// TIA Portal V15.1 export
// export: Created 2024-05-17T05:38:54.5333761Z, ExportSetting WithDefaults, DisplayName Totally Integrated Automation Portal, DisplayVersion V15.1 Update 5, DisplayName TIA Portal Openness, DisplayVersion V15.1 Update 5, DisplayName SINAMICS Startdrive Advanced, DisplayVersion V15.1, DisplayName G130, G150, S120, S150, SINAMICS MV, S210, DisplayVersion V15.1, DisplayName G110M, G120, G120C, G120D, G120P, DisplayVersion V15.1, DisplayName STEP 7 Professional, DisplayVersion V15.1 Update 5, DisplayName STEP 7 Safety, DisplayVersion V15.1, DisplayName WinCC Professional, DisplayVersion V15.1 Update 5, DisplayName SIMATIC Visualization Architect, DisplayVersion V15.1
FUNCTION "209220ZS01Passiv" : Void   // FC373, FBD
TITLE = 209220ZS01Passiv
{ S7_Optimized_Access := 'FALSE' }
AUTHOR : VCC
NAME : LocFunc
VERSION : 0.1
// stored: AutoNumber false, IsIECCheckEnabled false, SetENOAutomatically False, UDAEnableTagReadback false
   VAR_OUTPUT
      O_AlarmA : Bool;   // Alarm A
      O_AlarmB : Bool;   // Alarm B
      O_AlarmC : Bool;   // Alarm C
      O_AlarmD : Bool;   // Alarm D
      O_AlarmABCondition : Bool;   // Alarms resetable
      H_IAnim : Word;   // Icon Animation
   END_VAR
   VAR_TEMP
      TEMP0 : Bool;
   END_VAR
BEGIN

REGION Network 1: **** --------------------- ET200sp I/O --------------------- ****
END_REGION

REGION Network 2: **** 2.2 - Alarms - Alarm Generation **** 209000AK04JX37QF5270 - ET200sp I/O - Safety Card QF5270
   // Passivation alarm - ET200sp I/O - Safety Card QF5270
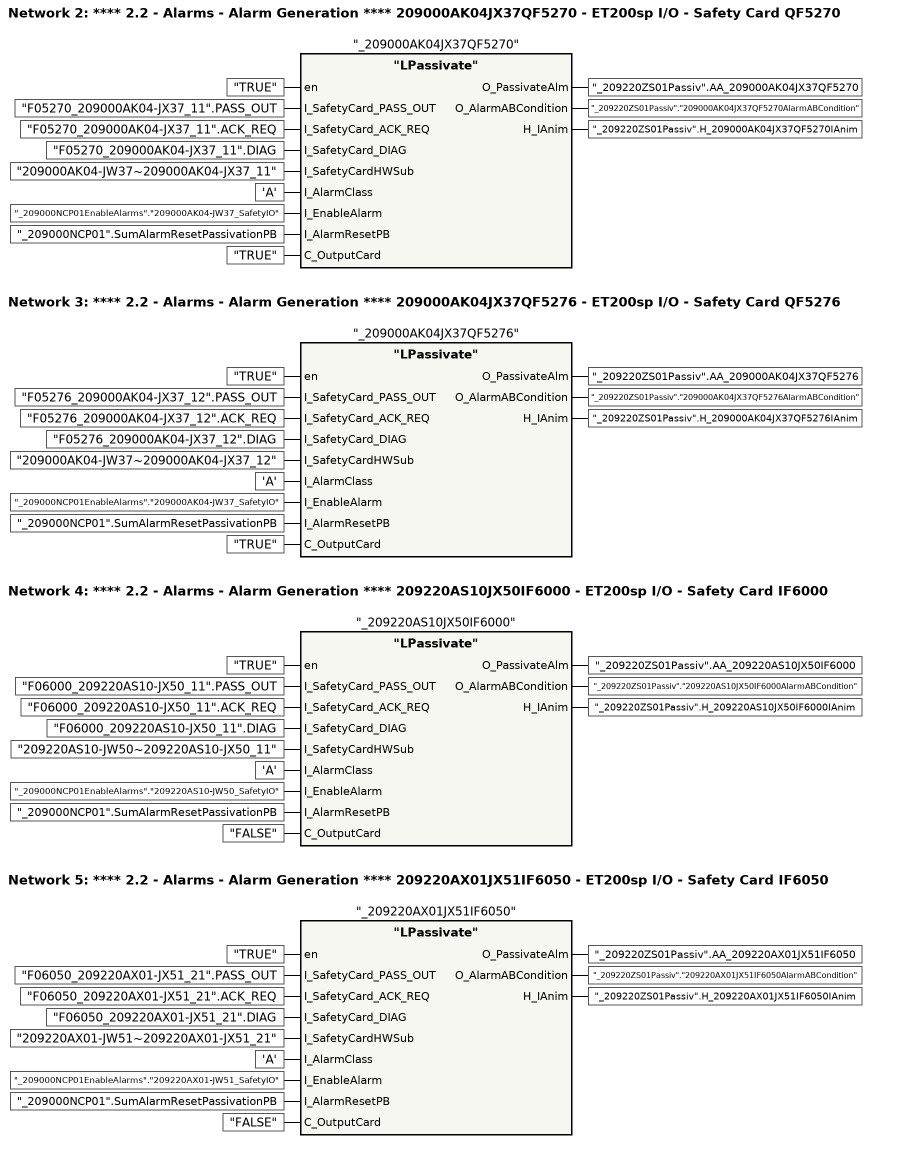
   IF "TRUE" THEN
       "_209000AK04JX37QF5270"(I_SafetyCard_PASS_OUT := "F05270_209000AK04-JX37_11".PASS_OUT,   // "LPassivate"
                               I_SafetyCard_ACK_REQ := "F05270_209000AK04-JX37_11".ACK_REQ,
                               I_SafetyCard_DIAG := "F05270_209000AK04-JX37_11".DIAG,
                               I_SafetyCardHWSub := "209000AK04-JW37~209000AK04-JX37_11",
                               I_AlarmClass := 'A',
                               I_EnableAlarm := "_209000NCP01EnableAlarms"."209000AK04-JW37_SafetyIO",
                               I_AlarmResetPB := "_209000NCP01".SumAlarmResetPassivationPB,
                               C_OutputCard := "TRUE",
                               O_PassivateAlm => "_209220ZS01Passiv".AA_209000AK04JX37QF5270,
                               O_AlarmABCondition => "_209220ZS01Passiv"."209000AK04JX37QF5270AlarmABCondition",
                               H_IAnim => "_209220ZS01Passiv".H_209000AK04JX37QF5270IAnim);
   END_IF;
END_REGION

REGION Network 3: **** 2.2 - Alarms - Alarm Generation **** 209000AK04JX37QF5276 - ET200sp I/O - Safety Card QF5276
   // Passivation alarm - ET200sp I/O - Safety Card QF5276
   IF "TRUE" THEN
       "_209000AK04JX37QF5276"(I_SafetyCard_PASS_OUT := "F05276_209000AK04-JX37_12".PASS_OUT,   // "LPassivate"
                               I_SafetyCard_ACK_REQ := "F05276_209000AK04-JX37_12".ACK_REQ,
                               I_SafetyCard_DIAG := "F05276_209000AK04-JX37_12".DIAG,
                               I_SafetyCardHWSub := "209000AK04-JW37~209000AK04-JX37_12",
                               I_AlarmClass := 'A',
                               I_EnableAlarm := "_209000NCP01EnableAlarms"."209000AK04-JW37_SafetyIO",
                               I_AlarmResetPB := "_209000NCP01".SumAlarmResetPassivationPB,
                               C_OutputCard := "TRUE",
                               O_PassivateAlm => "_209220ZS01Passiv".AA_209000AK04JX37QF5276,
                               O_AlarmABCondition => "_209220ZS01Passiv"."209000AK04JX37QF5276AlarmABCondition",
                               H_IAnim => "_209220ZS01Passiv".H_209000AK04JX37QF5276IAnim);
   END_IF;
END_REGION

REGION Network 4: **** 2.2 - Alarms - Alarm Generation **** 209220AS10JX50IF6000 - ET200sp I/O - Safety Card IF6000
   // Passivation alarm - ET200sp I/O - Safety Card IF6000
   IF "TRUE" THEN
       "_209220AS10JX50IF6000"(I_SafetyCard_PASS_OUT := "F06000_209220AS10-JX50_11".PASS_OUT,   // "LPassivate"
                               I_SafetyCard_ACK_REQ := "F06000_209220AS10-JX50_11".ACK_REQ,
                               I_SafetyCard_DIAG := "F06000_209220AS10-JX50_11".DIAG,
                               I_SafetyCardHWSub := "209220AS10-JW50~209220AS10-JX50_11",
                               I_AlarmClass := 'A',
                               I_EnableAlarm := "_209000NCP01EnableAlarms"."209220AS10-JW50_SafetyIO",
                               I_AlarmResetPB := "_209000NCP01".SumAlarmResetPassivationPB,
                               C_OutputCard := "FALSE",
                               O_PassivateAlm => "_209220ZS01Passiv".AA_209220AS10JX50IF6000,
                               O_AlarmABCondition => "_209220ZS01Passiv"."209220AS10JX50IF6000AlarmABCondition",
                               H_IAnim => "_209220ZS01Passiv".H_209220AS10JX50IF6000IAnim);
   END_IF;
END_REGION

REGION Network 5: **** 2.2 - Alarms - Alarm Generation **** 209220AX01JX51IF6050 - ET200sp I/O - Safety Card IF6050
   // Passivation alarm - ET200sp I/O - Safety Card IF6050
   IF "TRUE" THEN
       "_209220AX01JX51IF6050"(I_SafetyCard_PASS_OUT := "F06050_209220AX01-JX51_21".PASS_OUT,   // "LPassivate"
                               I_SafetyCard_ACK_REQ := "F06050_209220AX01-JX51_21".ACK_REQ,
                               I_SafetyCard_DIAG := "F06050_209220AX01-JX51_21".DIAG,
                               I_SafetyCardHWSub := "209220AX01-JW51~209220AX01-JX51_21",
                               I_AlarmClass := 'A',
                               I_EnableAlarm := "_209000NCP01EnableAlarms"."209220AX01-JW51_SafetyIO",
                               I_AlarmResetPB := "_209000NCP01".SumAlarmResetPassivationPB,
                               C_OutputCard := "FALSE",
                               O_PassivateAlm => "_209220ZS01Passiv".AA_209220AX01JX51IF6050,
                               O_AlarmABCondition => "_209220ZS01Passiv"."209220AX01JX51IF6050AlarmABCondition",
                               H_IAnim => "_209220ZS01Passiv".H_209220AX01JX51IF6050IAnim);
   END_IF;
END_REGION

REGION Network 6: **** 2.2 - Alarms - Alarm Generation **** 209220AS11JX52IF6100 - ET200sp I/O - Safety Card IF6100
   // Passivation alarm - ET200sp I/O - Safety Card IF6100
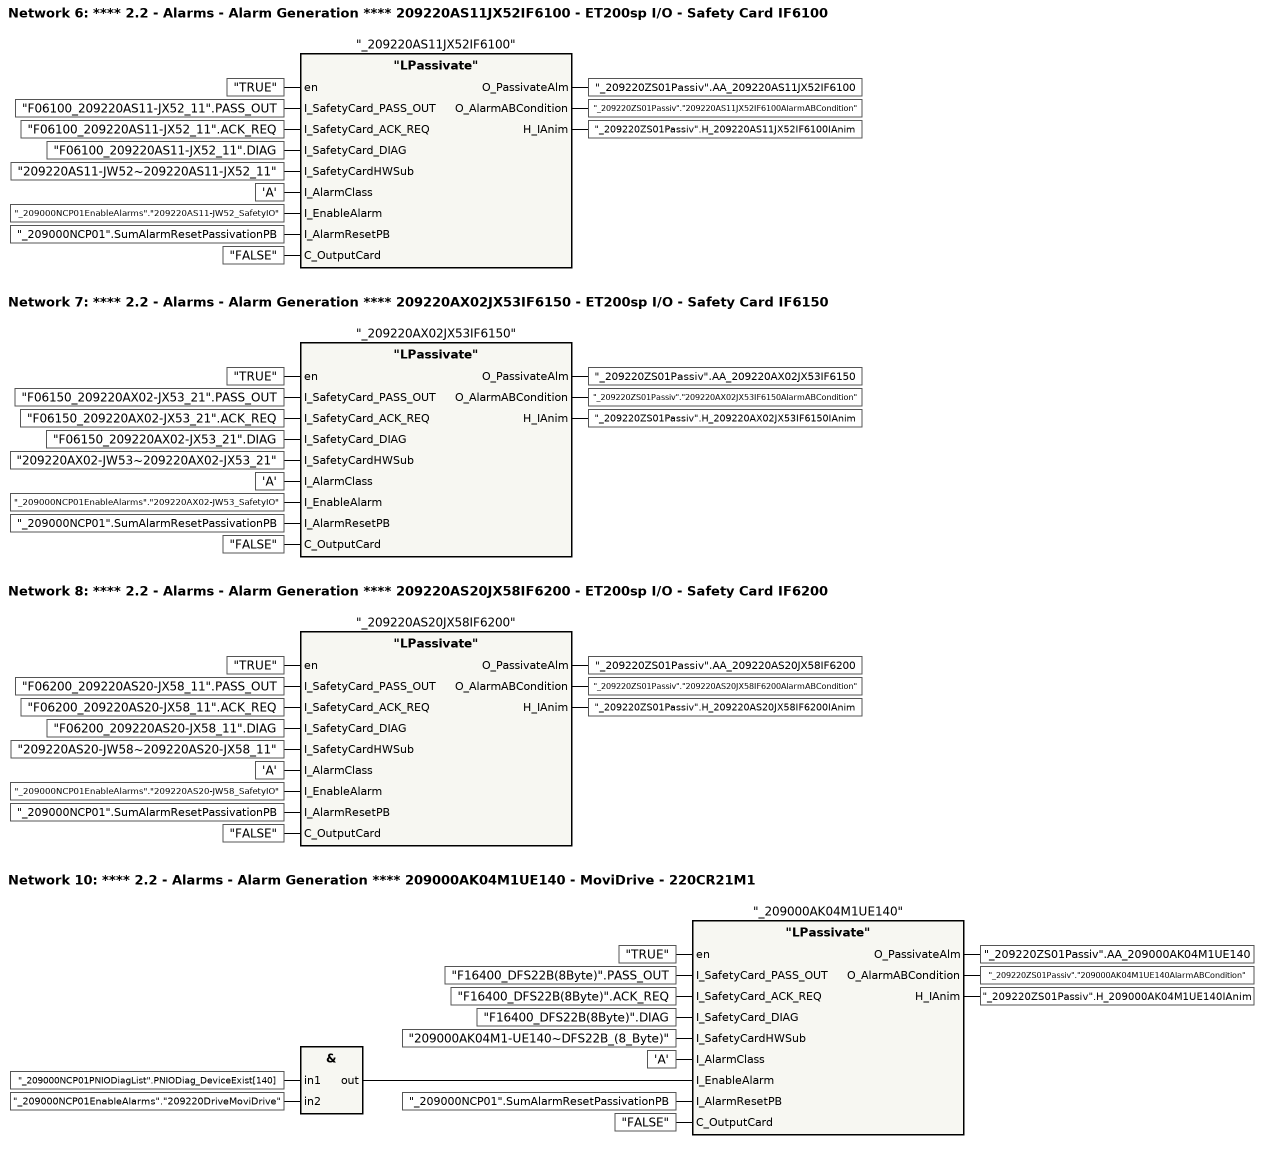
   IF "TRUE" THEN
       "_209220AS11JX52IF6100"(I_SafetyCard_PASS_OUT := "F06100_209220AS11-JX52_11".PASS_OUT,   // "LPassivate"
                               I_SafetyCard_ACK_REQ := "F06100_209220AS11-JX52_11".ACK_REQ,
                               I_SafetyCard_DIAG := "F06100_209220AS11-JX52_11".DIAG,
                               I_SafetyCardHWSub := "209220AS11-JW52~209220AS11-JX52_11",
                               I_AlarmClass := 'A',
                               I_EnableAlarm := "_209000NCP01EnableAlarms"."209220AS11-JW52_SafetyIO",
                               I_AlarmResetPB := "_209000NCP01".SumAlarmResetPassivationPB,
                               C_OutputCard := "FALSE",
                               O_PassivateAlm => "_209220ZS01Passiv".AA_209220AS11JX52IF6100,
                               O_AlarmABCondition => "_209220ZS01Passiv"."209220AS11JX52IF6100AlarmABCondition",
                               H_IAnim => "_209220ZS01Passiv".H_209220AS11JX52IF6100IAnim);
   END_IF;
END_REGION

REGION Network 7: **** 2.2 - Alarms - Alarm Generation **** 209220AX02JX53IF6150 - ET200sp I/O - Safety Card IF6150
   // Passivation alarm - ET200sp I/O - Safety Card IF6150
   IF "TRUE" THEN
       "_209220AX02JX53IF6150"(I_SafetyCard_PASS_OUT := "F06150_209220AX02-JX53_21".PASS_OUT,   // "LPassivate"
                               I_SafetyCard_ACK_REQ := "F06150_209220AX02-JX53_21".ACK_REQ,
                               I_SafetyCard_DIAG := "F06150_209220AX02-JX53_21".DIAG,
                               I_SafetyCardHWSub := "209220AX02-JW53~209220AX02-JX53_21",
                               I_AlarmClass := 'A',
                               I_EnableAlarm := "_209000NCP01EnableAlarms"."209220AX02-JW53_SafetyIO",
                               I_AlarmResetPB := "_209000NCP01".SumAlarmResetPassivationPB,
                               C_OutputCard := "FALSE",
                               O_PassivateAlm => "_209220ZS01Passiv".AA_209220AX02JX53IF6150,
                               O_AlarmABCondition => "_209220ZS01Passiv"."209220AX02JX53IF6150AlarmABCondition",
                               H_IAnim => "_209220ZS01Passiv".H_209220AX02JX53IF6150IAnim);
   END_IF;
END_REGION

REGION Network 8: **** 2.2 - Alarms - Alarm Generation **** 209220AS20JX58IF6200 - ET200sp I/O - Safety Card IF6200
   // Passivation alarm - ET200sp I/O - Safety Card IF6200
   IF "TRUE" THEN
       "_209220AS20JX58IF6200"(I_SafetyCard_PASS_OUT := "F06200_209220AS20-JX58_11".PASS_OUT,   // "LPassivate"
                               I_SafetyCard_ACK_REQ := "F06200_209220AS20-JX58_11".ACK_REQ,
                               I_SafetyCard_DIAG := "F06200_209220AS20-JX58_11".DIAG,
                               I_SafetyCardHWSub := "209220AS20-JW58~209220AS20-JX58_11",
                               I_AlarmClass := 'A',
                               I_EnableAlarm := "_209000NCP01EnableAlarms"."209220AS20-JW58_SafetyIO",
                               I_AlarmResetPB := "_209000NCP01".SumAlarmResetPassivationPB,
                               C_OutputCard := "FALSE",
                               O_PassivateAlm => "_209220ZS01Passiv".AA_209220AS20JX58IF6200,
                               O_AlarmABCondition => "_209220ZS01Passiv"."209220AS20JX58IF6200AlarmABCondition",
                               H_IAnim => "_209220ZS01Passiv".H_209220AS20JX58IF6200IAnim);
   END_IF;
END_REGION

REGION Network 9: **** --------------------- Drive --------------------- ****
END_REGION

REGION Network 10: **** 2.2 - Alarms - Alarm Generation **** 209000AK04M1UE140 - MoviDrive - 220CR21M1
   // Passivation alarm - MoviDrive - 220CR21M1
   IF "TRUE" THEN
       "_209000AK04M1UE140"(I_SafetyCard_PASS_OUT := "F16400_DFS22B(8Byte)".PASS_OUT,   // "LPassivate"
                            I_SafetyCard_ACK_REQ := "F16400_DFS22B(8Byte)".ACK_REQ,
                            I_SafetyCard_DIAG := "F16400_DFS22B(8Byte)".DIAG,
                            I_SafetyCardHWSub := "209000AK04M1-UE140~DFS22B_(8_Byte)",
                            I_AlarmClass := 'A',
                            I_EnableAlarm := "_209000NCP01PNIODiagList".PNIODiag_DeviceExist[140] AND "_209000NCP01EnableAlarms"."209220DriveMoviDrive",
                            I_AlarmResetPB := "_209000NCP01".SumAlarmResetPassivationPB,
                            C_OutputCard := "FALSE",
                            O_PassivateAlm => "_209220ZS01Passiv".AA_209000AK04M1UE140,
                            O_AlarmABCondition => "_209220ZS01Passiv"."209000AK04M1UE140AlarmABCondition",
                            H_IAnim => "_209220ZS01Passiv".H_209000AK04M1UE140IAnim);
   END_IF;
END_REGION

REGION Network 11: **** 2.2 - Alarms - Alarm Generation **** 209000AK04M4UE141 - MoviDrive - 220CS22M4ME1 (Power)
   // Passivation alarm - MoviDrive - 220CS22M4ME1 (Power)
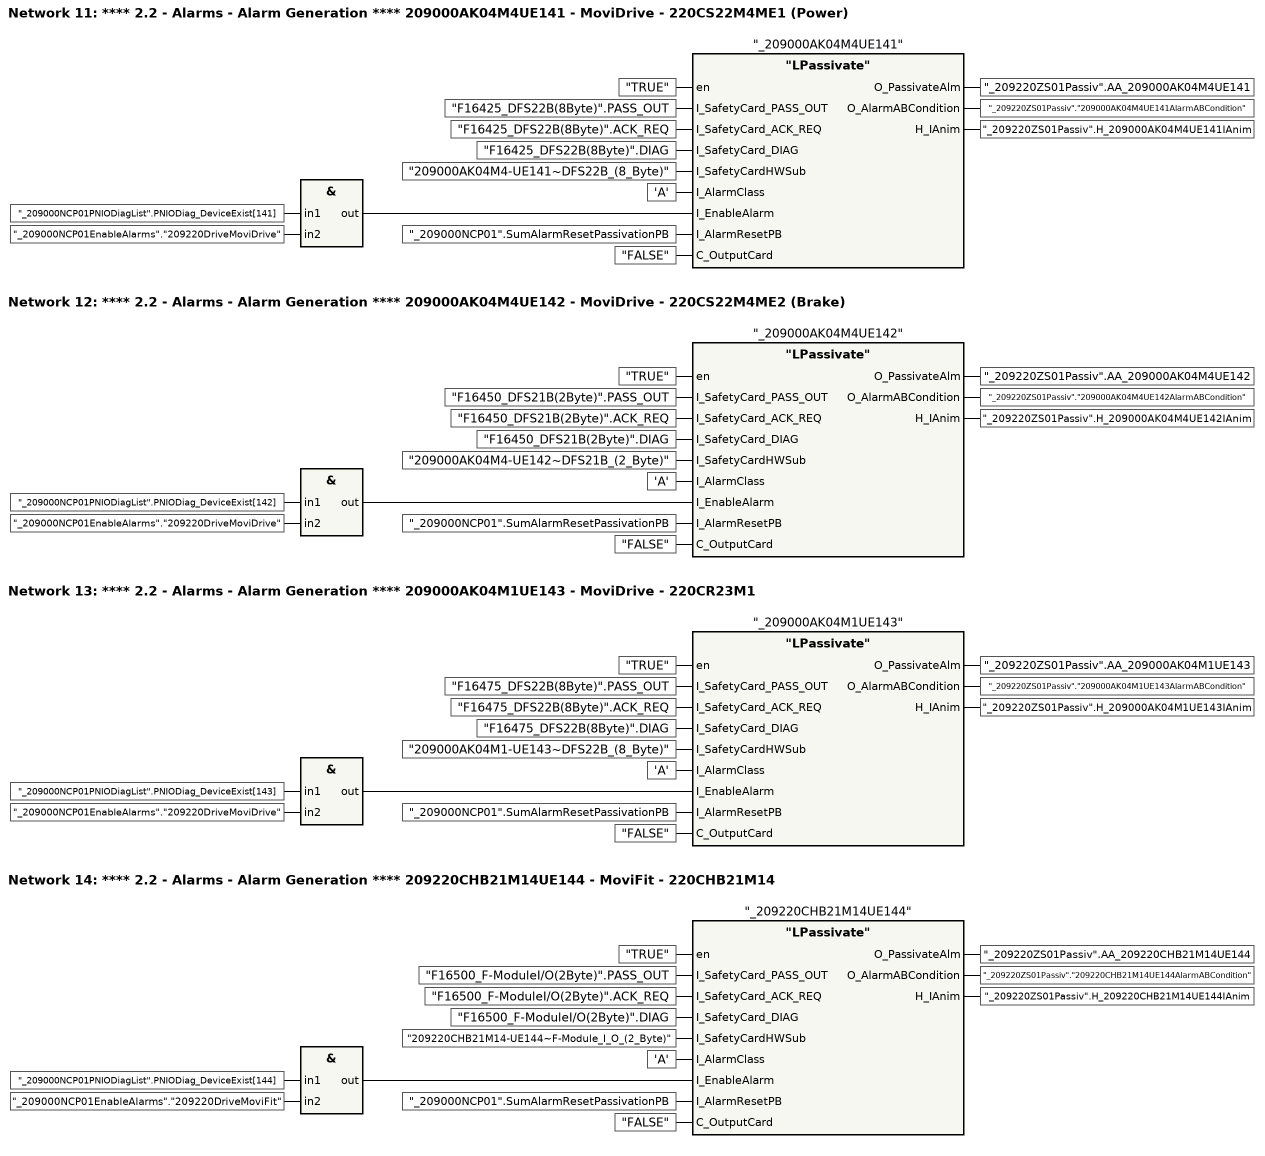
   IF "TRUE" THEN
       "_209000AK04M4UE141"(I_SafetyCard_PASS_OUT := "F16425_DFS22B(8Byte)".PASS_OUT,   // "LPassivate"
                            I_SafetyCard_ACK_REQ := "F16425_DFS22B(8Byte)".ACK_REQ,
                            I_SafetyCard_DIAG := "F16425_DFS22B(8Byte)".DIAG,
                            I_SafetyCardHWSub := "209000AK04M4-UE141~DFS22B_(8_Byte)",
                            I_AlarmClass := 'A',
                            I_EnableAlarm := "_209000NCP01PNIODiagList".PNIODiag_DeviceExist[141] AND "_209000NCP01EnableAlarms"."209220DriveMoviDrive",
                            I_AlarmResetPB := "_209000NCP01".SumAlarmResetPassivationPB,
                            C_OutputCard := "FALSE",
                            O_PassivateAlm => "_209220ZS01Passiv".AA_209000AK04M4UE141,
                            O_AlarmABCondition => "_209220ZS01Passiv"."209000AK04M4UE141AlarmABCondition",
                            H_IAnim => "_209220ZS01Passiv".H_209000AK04M4UE141IAnim);
   END_IF;
END_REGION

REGION Network 12: **** 2.2 - Alarms - Alarm Generation **** 209000AK04M4UE142 - MoviDrive - 220CS22M4ME2 (Brake)
   // Passivation alarm - MoviDrive - 220CS22M4ME2 (Brake)
   IF "TRUE" THEN
       "_209000AK04M4UE142"(I_SafetyCard_PASS_OUT := "F16450_DFS21B(2Byte)".PASS_OUT,   // "LPassivate"
                            I_SafetyCard_ACK_REQ := "F16450_DFS21B(2Byte)".ACK_REQ,
                            I_SafetyCard_DIAG := "F16450_DFS21B(2Byte)".DIAG,
                            I_SafetyCardHWSub := "209000AK04M4-UE142~DFS21B_(2_Byte)",
                            I_AlarmClass := 'A',
                            I_EnableAlarm := "_209000NCP01PNIODiagList".PNIODiag_DeviceExist[142] AND "_209000NCP01EnableAlarms"."209220DriveMoviDrive",
                            I_AlarmResetPB := "_209000NCP01".SumAlarmResetPassivationPB,
                            C_OutputCard := "FALSE",
                            O_PassivateAlm => "_209220ZS01Passiv".AA_209000AK04M4UE142,
                            O_AlarmABCondition => "_209220ZS01Passiv"."209000AK04M4UE142AlarmABCondition",
                            H_IAnim => "_209220ZS01Passiv".H_209000AK04M4UE142IAnim);
   END_IF;
END_REGION

REGION Network 13: **** 2.2 - Alarms - Alarm Generation **** 209000AK04M1UE143 - MoviDrive - 220CR23M1
   // Passivation alarm - MoviDrive - 220CR23M1
   IF "TRUE" THEN
       "_209000AK04M1UE143"(I_SafetyCard_PASS_OUT := "F16475_DFS22B(8Byte)".PASS_OUT,   // "LPassivate"
                            I_SafetyCard_ACK_REQ := "F16475_DFS22B(8Byte)".ACK_REQ,
                            I_SafetyCard_DIAG := "F16475_DFS22B(8Byte)".DIAG,
                            I_SafetyCardHWSub := "209000AK04M1-UE143~DFS22B_(8_Byte)",
                            I_AlarmClass := 'A',
                            I_EnableAlarm := "_209000NCP01PNIODiagList".PNIODiag_DeviceExist[143] AND "_209000NCP01EnableAlarms"."209220DriveMoviDrive",
                            I_AlarmResetPB := "_209000NCP01".SumAlarmResetPassivationPB,
                            C_OutputCard := "FALSE",
                            O_PassivateAlm => "_209220ZS01Passiv".AA_209000AK04M1UE143,
                            O_AlarmABCondition => "_209220ZS01Passiv"."209000AK04M1UE143AlarmABCondition",
                            H_IAnim => "_209220ZS01Passiv".H_209000AK04M1UE143IAnim);
   END_IF;
END_REGION

REGION Network 14: **** 2.2 - Alarms - Alarm Generation **** 209220CHB21M14UE144 - MoviFit - 220CHB21M14
   // Passivation alarm - MoviFit - 220CHB21M14
   IF "TRUE" THEN
       "_209220CHB21M14UE144"(I_SafetyCard_PASS_OUT := "F16500_F-ModuleI/O(2Byte)".PASS_OUT,   // "LPassivate"
                              I_SafetyCard_ACK_REQ := "F16500_F-ModuleI/O(2Byte)".ACK_REQ,
                              I_SafetyCard_DIAG := "F16500_F-ModuleI/O(2Byte)".DIAG,
                              I_SafetyCardHWSub := "209220CHB21M14-UE144~F-Module_I_O_(2_Byte)",
                              I_AlarmClass := 'A',
                              I_EnableAlarm := "_209000NCP01PNIODiagList".PNIODiag_DeviceExist[144] AND "_209000NCP01EnableAlarms"."209220DriveMoviFit",
                              I_AlarmResetPB := "_209000NCP01".SumAlarmResetPassivationPB,
                              C_OutputCard := "FALSE",
                              O_PassivateAlm => "_209220ZS01Passiv".AA_209220CHB21M14UE144,
                              O_AlarmABCondition => "_209220ZS01Passiv"."209220CHB21M14UE144AlarmABCondition",
                              H_IAnim => "_209220ZS01Passiv".H_209220CHB21M14UE144IAnim);
   END_IF;
END_REGION

REGION Network 15: **** -------------------------------------------------- ****
END_REGION

REGION Network 16: **** 4.6 - Machine Status - Indications **** Icon animation
   // Icon animation
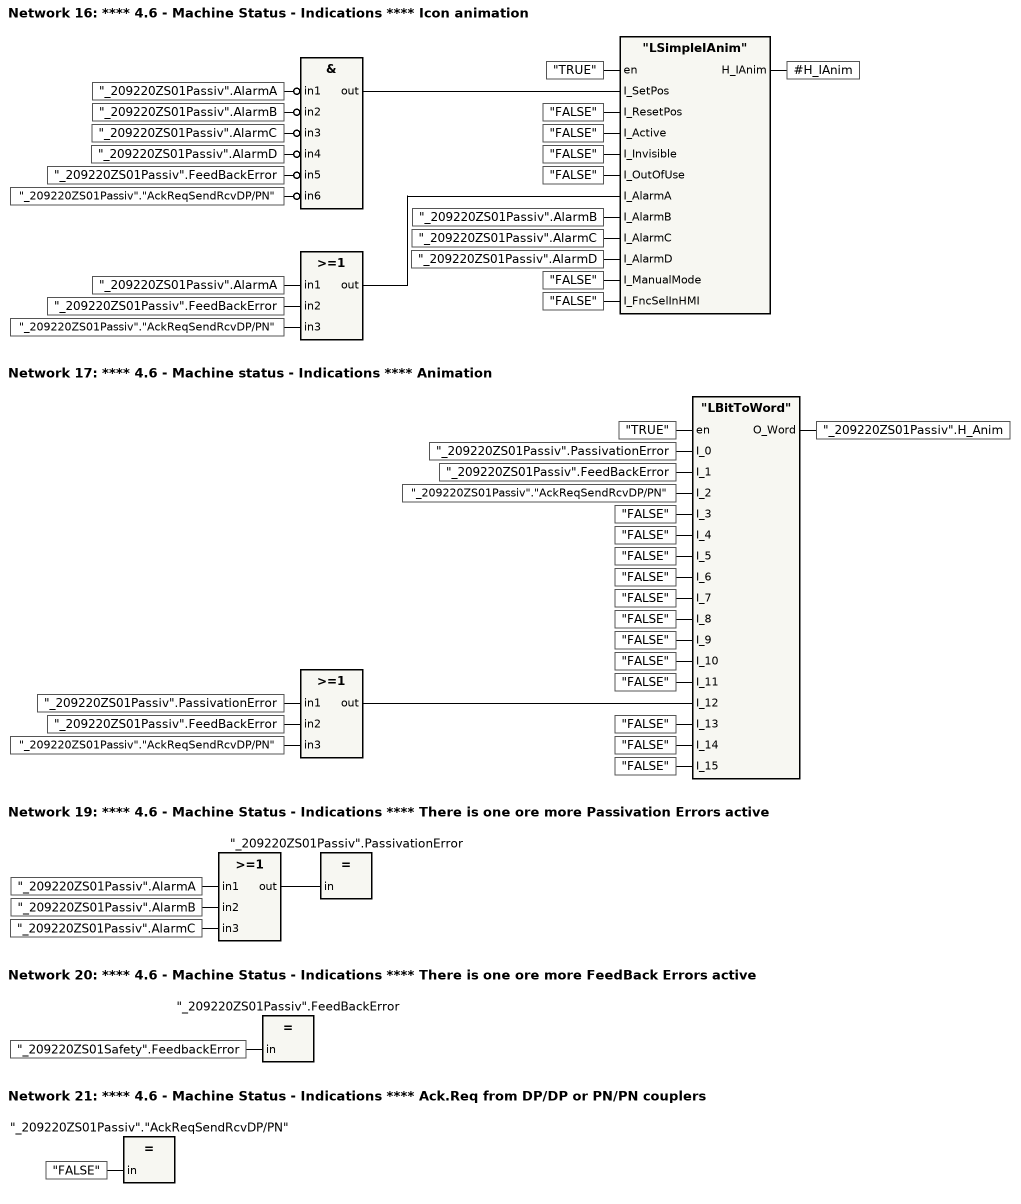
   IF "TRUE" THEN
       "LSimpleIAnim"(I_SetPos := NOT "_209220ZS01Passiv".AlarmA AND NOT "_209220ZS01Passiv".AlarmB AND NOT "_209220ZS01Passiv".AlarmC AND NOT "_209220ZS01Passiv".AlarmD AND NOT "_209220ZS01Passiv".FeedBackError AND NOT "_209220ZS01Passiv"."AckReqSendRcvDP/PN",
                      I_ResetPos := "FALSE",
                      I_Active := "FALSE",
                      I_Invisible := "FALSE",
                      I_OutOfUse := "FALSE",
                      I_AlarmA := "_209220ZS01Passiv".AlarmA OR "_209220ZS01Passiv".FeedBackError OR "_209220ZS01Passiv"."AckReqSendRcvDP/PN",
                      I_AlarmB := "_209220ZS01Passiv".AlarmB,
                      I_AlarmC := "_209220ZS01Passiv".AlarmC,
                      I_AlarmD := "_209220ZS01Passiv".AlarmD,
                      I_ManualMode := "FALSE",
                      I_FncSelInHMI := "FALSE",
                      H_IAnim => #H_IAnim);
   END_IF;
END_REGION

REGION Network 17: **** 4.6 - Machine status - Indications **** Animation
   // Animation
   IF "TRUE" THEN
       "LBitToWord"(I_0 := "_209220ZS01Passiv".PassivationError,
                    I_1 := "_209220ZS01Passiv".FeedBackError,
                    I_2 := "_209220ZS01Passiv"."AckReqSendRcvDP/PN",
                    I_3 := "FALSE",
                    I_4 := "FALSE",
                    I_5 := "FALSE",
                    I_6 := "FALSE",
                    I_7 := "FALSE",
                    I_8 := "FALSE",
                    I_9 := "FALSE",
                    I_10 := "FALSE",
                    I_11 := "FALSE",
                    I_12 := "_209220ZS01Passiv".PassivationError OR "_209220ZS01Passiv".FeedBackError OR "_209220ZS01Passiv"."AckReqSendRcvDP/PN",
                    I_13 := "FALSE",
                    I_14 := "FALSE",
                    I_15 := "FALSE",
                    O_Word => "_209220ZS01Passiv".H_Anim);
   END_IF;
END_REGION

NETWORK
TITLE = **** 4.6 - Machine Status - Indications **** Animation DB number
// DB number
      OPN   "_209220ZS01Passiv";
      L     DBNO;
      T     "_209220ZS01Passiv".H_DBnr;

REGION Network 19: **** 4.6 - Machine Status - Indications **** There is one ore more Passivation Errors active
   // There is one ore more Passivation Errors active
   "_209220ZS01Passiv".PassivationError := "_209220ZS01Passiv".AlarmA OR "_209220ZS01Passiv".AlarmB OR "_209220ZS01Passiv".AlarmC;
END_REGION

REGION Network 20: **** 4.6 - Machine Status - Indications **** There is one ore more FeedBack Errors active
   // There is one ore more FeedBack Errors active
   "_209220ZS01Passiv".FeedBackError := "_209220ZS01Safety".FeedbackError;
END_REGION

REGION Network 21: **** 4.6 - Machine Status - Indications **** Ack.Req from DP/DP or PN/PN couplers
   // Ack.Req from DP/DP or PN/PN couplers
   "_209220ZS01Passiv"."AckReqSendRcvDP/PN" := "FALSE";
END_REGION

REGION Network 22: **** 9 - Alarm Summary **** Alarm AB Condition
   // Alarm AB condition
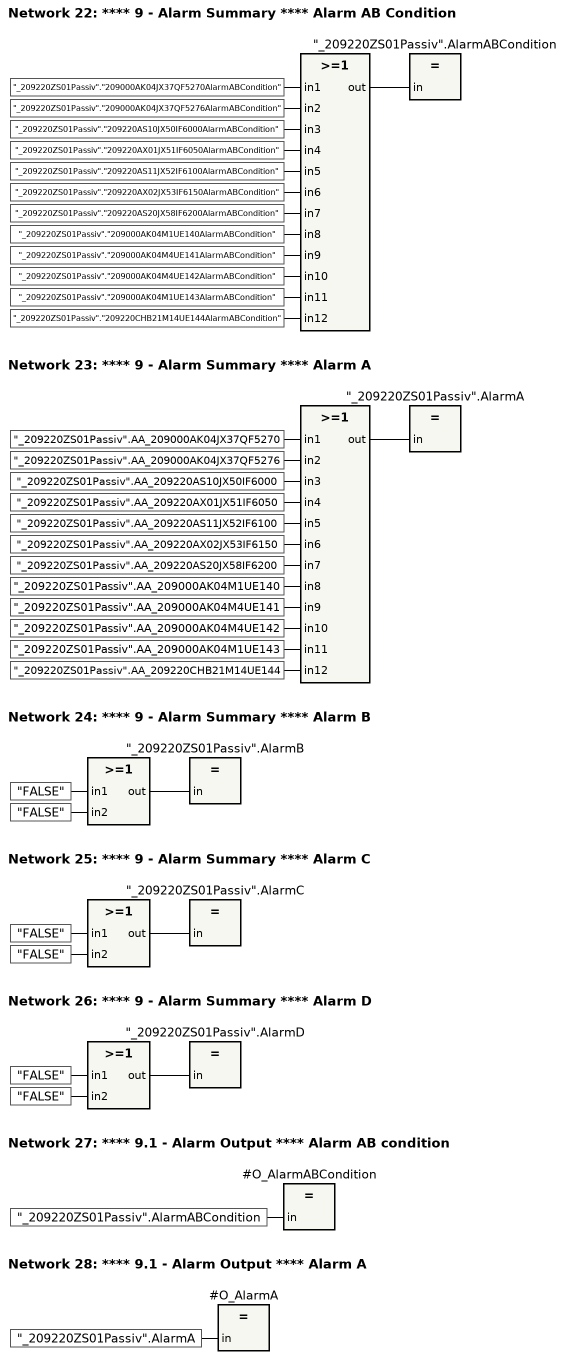
   "_209220ZS01Passiv".AlarmABCondition := "_209220ZS01Passiv"."209000AK04JX37QF5270AlarmABCondition" OR "_209220ZS01Passiv"."209000AK04JX37QF5276AlarmABCondition" OR "_209220ZS01Passiv"."209220AS10JX50IF6000AlarmABCondition" OR "_209220ZS01Passiv"."209220AX01JX51IF6050AlarmABCondition" OR "_209220ZS01Passiv"."209220AS11JX52IF6100AlarmABCondition" OR "_209220ZS01Passiv"."209220AX02JX53IF6150AlarmABCondition" OR "_209220ZS01Passiv"."209220AS20JX58IF6200AlarmABCondition" OR "_209220ZS01Passiv"."209000AK04M1UE140AlarmABCondition" OR "_209220ZS01Passiv"."209000AK04M4UE141AlarmABCondition" OR "_209220ZS01Passiv"."209000AK04M4UE142AlarmABCondition" OR "_209220ZS01Passiv"."209000AK04M1UE143AlarmABCondition" OR "_209220ZS01Passiv"."209220CHB21M14UE144AlarmABCondition";
END_REGION

REGION Network 23: **** 9 - Alarm Summary **** Alarm A
   // Summary of alarms A
   "_209220ZS01Passiv".AlarmA := "_209220ZS01Passiv".AA_209000AK04JX37QF5270 OR "_209220ZS01Passiv".AA_209000AK04JX37QF5276 OR "_209220ZS01Passiv".AA_209220AS10JX50IF6000 OR "_209220ZS01Passiv".AA_209220AX01JX51IF6050 OR "_209220ZS01Passiv".AA_209220AS11JX52IF6100 OR "_209220ZS01Passiv".AA_209220AX02JX53IF6150 OR "_209220ZS01Passiv".AA_209220AS20JX58IF6200 OR "_209220ZS01Passiv".AA_209000AK04M1UE140 OR "_209220ZS01Passiv".AA_209000AK04M4UE141 OR "_209220ZS01Passiv".AA_209000AK04M4UE142 OR "_209220ZS01Passiv".AA_209000AK04M1UE143 OR "_209220ZS01Passiv".AA_209220CHB21M14UE144;
END_REGION

REGION Network 24: **** 9 - Alarm Summary **** Alarm B
   // Summary of alarms B
   "_209220ZS01Passiv".AlarmB := "FALSE" OR "FALSE";
END_REGION

REGION Network 25: **** 9 - Alarm Summary **** Alarm C
   // Summary of alarms C
   "_209220ZS01Passiv".AlarmC := "FALSE" OR "FALSE";
END_REGION

REGION Network 26: **** 9 - Alarm Summary **** Alarm D
   // Summary of alarms D
   "_209220ZS01Passiv".AlarmD := "FALSE" OR "FALSE";
END_REGION

REGION Network 27: **** 9.1 - Alarm Output **** Alarm AB condition
   // Alarm AB condition
   #O_AlarmABCondition := "_209220ZS01Passiv".AlarmABCondition;
END_REGION

REGION Network 28: **** 9.1 - Alarm Output **** Alarm A
   // Output Alarm A
   #O_AlarmA := "_209220ZS01Passiv".AlarmA;
END_REGION

REGION Network 29: **** 9.1 - Alarm Output **** Alarm B
   // Output Alarm B
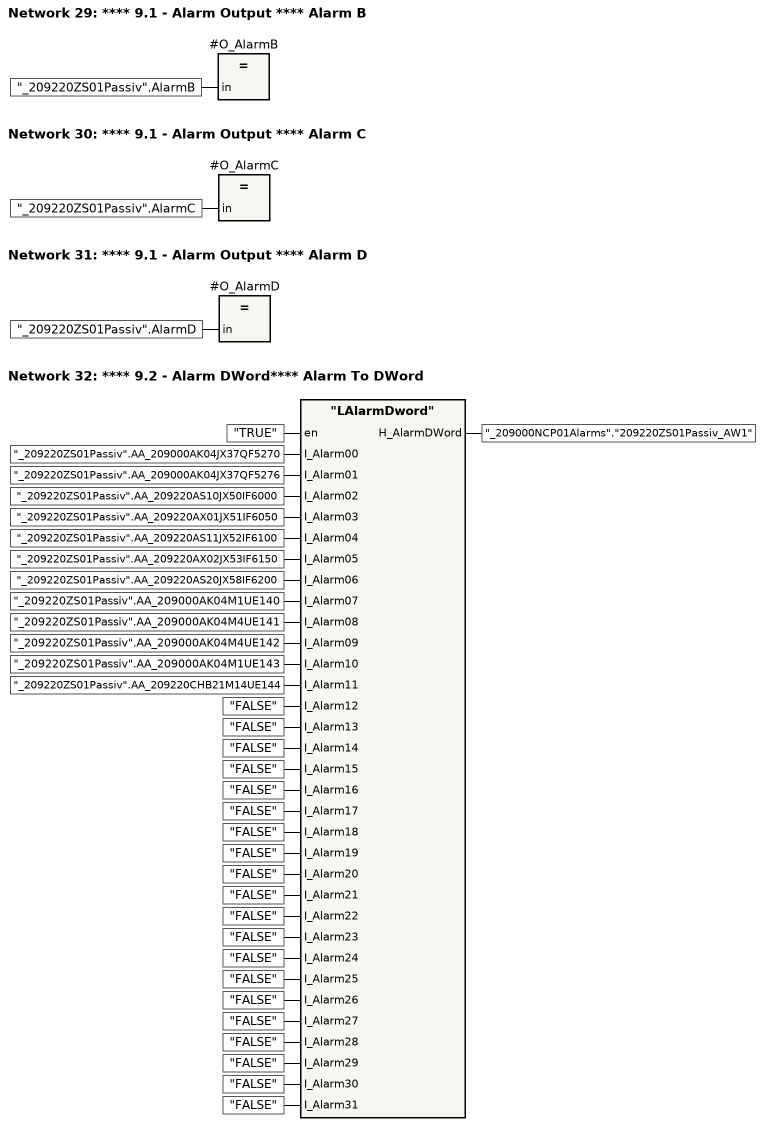
   #O_AlarmB := "_209220ZS01Passiv".AlarmB;
END_REGION

REGION Network 30: **** 9.1 - Alarm Output **** Alarm C
   // Output Alarm C
   #O_AlarmC := "_209220ZS01Passiv".AlarmC;
END_REGION

REGION Network 31: **** 9.1 - Alarm Output **** Alarm D
   // Output Alarm D
   #O_AlarmD := "_209220ZS01Passiv".AlarmD;
END_REGION

REGION Network 32: **** 9.2 - Alarm DWord**** Alarm To DWord
   // Alarm Word
   IF "TRUE" THEN
       "LAlarmDword"(I_Alarm00 := "_209220ZS01Passiv".AA_209000AK04JX37QF5270,
                     I_Alarm01 := "_209220ZS01Passiv".AA_209000AK04JX37QF5276,
                     I_Alarm02 := "_209220ZS01Passiv".AA_209220AS10JX50IF6000,
                     I_Alarm03 := "_209220ZS01Passiv".AA_209220AX01JX51IF6050,
                     I_Alarm04 := "_209220ZS01Passiv".AA_209220AS11JX52IF6100,
                     I_Alarm05 := "_209220ZS01Passiv".AA_209220AX02JX53IF6150,
                     I_Alarm06 := "_209220ZS01Passiv".AA_209220AS20JX58IF6200,
                     I_Alarm07 := "_209220ZS01Passiv".AA_209000AK04M1UE140,
                     I_Alarm08 := "_209220ZS01Passiv".AA_209000AK04M4UE141,
                     I_Alarm09 := "_209220ZS01Passiv".AA_209000AK04M4UE142,
                     I_Alarm10 := "_209220ZS01Passiv".AA_209000AK04M1UE143,
                     I_Alarm11 := "_209220ZS01Passiv".AA_209220CHB21M14UE144,
                     I_Alarm12 := "FALSE",
                     I_Alarm13 := "FALSE",
                     I_Alarm14 := "FALSE",
                     I_Alarm15 := "FALSE",
                     I_Alarm16 := "FALSE",
                     I_Alarm17 := "FALSE",
                     I_Alarm18 := "FALSE",
                     I_Alarm19 := "FALSE",
                     I_Alarm20 := "FALSE",
                     I_Alarm21 := "FALSE",
                     I_Alarm22 := "FALSE",
                     I_Alarm23 := "FALSE",
                     I_Alarm24 := "FALSE",
                     I_Alarm25 := "FALSE",
                     I_Alarm26 := "FALSE",
                     I_Alarm27 := "FALSE",
                     I_Alarm28 := "FALSE",
                     I_Alarm29 := "FALSE",
                     I_Alarm30 := "FALSE",
                     I_Alarm31 := "FALSE",
                     H_AlarmDWord => "_209000NCP01Alarms"."209220ZS01Passiv_AW1");
   END_IF;
END_REGION
END_FUNCTION
